{attribute 'strict'}
{attribute 'to_string'}
TYPE MainStateMachine_enum :
(
	MS_DISABLED			:= 0,
	MS_INITIALIZING		:= 10,
	MS_ENABLED			:= 20,
	MS_RUN				:= 30,
	MS_STOPPING			:= 40,
	MS_STOPPED			:= 50,
	MS_DISABLING		:= 60,
	MS_ERROR			:= 70,
	MS_DEBUG			:= 80	
);
END_TYPE

(* stored: Version 1.1.0.1, ProductVersion 3.1.4026.8
   DUT MainStateMachine_enum: Id {95d9048c-947b-0f01-3cd5-5e396a74ec2a} *)
